TYPE mcInterface :
STRUCT
	bBusy				: BOOL;
	bActive				: BOOL;
	bCommandAborted		: BOOL;
	bError				: BOOL;
	iErrorID			: UDINT;
END_STRUCT
END_TYPE

(* stored: Version 1.1.0.1, ProductVersion 3.1.4024.12
   DUT mcInterface: Id {83da3ce5-8cbb-49d7-92f7-4a9709920a37} *)
